// TIA Portal V19 program export: 2 tag tables, 0 data types, 0 data blocks, 5 code blocks (in call order from the OBs), 7 instance data blocks

VAR_GLOBAL   // PLC tag table "Default tag table"
   Sensor_High_High AT %M0.0 : Bool;
   ACK_Alarm_PB AT %M0.1 : Bool;
   Alarm_Reset_PB AT %M0.2 : Bool;
   AlarmStatus AT %M0.3 : Bool;
   Alarm_Acknowledged AT %M0.4 : Bool;
   Alarm_LED AT %M0.5 : Bool;
   Sensor2_High_High AT %M1.0 : Bool;
   AlarmStatus2 AT %M1.1 : Bool;
   Alarm_Acknowledged2 AT %M0.6 : Bool;
   Alarm_LED2 AT %M0.7 : Bool;
END_VAR

VAR_GLOBAL   // PLC tag table "Dispenser_Tags"
   Power_ON AT %M1.0 : Bool;   // Power on Command
   Power_OFF AT %M1.1 : Bool;   // Power off Command
   Power_Active AT %M1.2 : Bool;   // Power is Active
   Start AT %M1.3 : Bool;   // Start Command
   Motor AT %M1.5 : Bool;   // Motor Status
   Gate1 AT %M1.6 : Bool;   // Light Gate Sensor 1
   Gate2 AT %M1.7 : Bool;   // Light Gate Sensor 2
   Gate3 AT %M2.0 : Bool;   // Light Gate Sensor 3
   Gate4 AT %M2.1 : Bool;   // Light Gate Sensor 4
   Gate5 AT %M2.2 : Bool;   // Light Gate Sensor 5
   Dropper_A AT %M2.3 : Bool;   // Dispenser Dropper 1
   Dropper_B AT %M2.4 : Bool;   // Dispenser Dropper 2
   Dropper_C AT %M2.5 : Bool;   // Dispenser Dropper 3
   Stop AT %M1.4 : Bool;   // Stop Command
   SW_A AT %M2.6 : Bool;   // Switch A
   SW_B AT %M2.7 : Bool;   // Switch B
   SW_C AT %M3.0 : Bool;   // Switch C
   Process_Started AT %M3.1 : Bool;   // Dispenser Process Running
   StopDispenser AT %M3.2 : Bool;   // E-Stop for Dispenser
END_VAR

ORGANIZATION_BLOCK "Main"   // OB1, LAD, ProgramCycle
TITLE = "Main Program Sweep (Cycle)"
{ S7_Optimized_Access := 'TRUE' }
// stored: SetENOAutomatically false
   VAR_INPUT
      Initial_Call : Bool;   // Initial call of this OB
      Remanence : Bool;   // =True, if remanent data are available
   END_VAR
BEGIN

REGION Network 1: Sensor 1 - Alarm
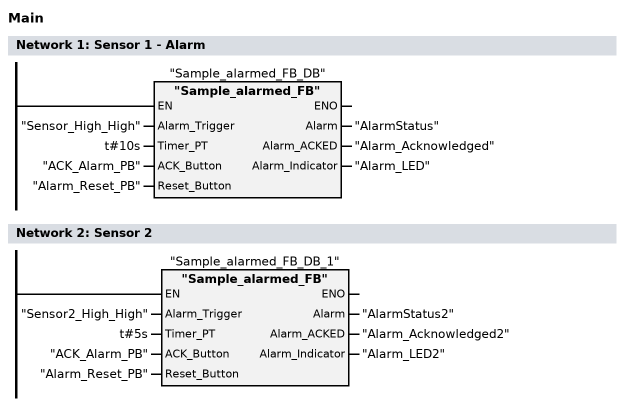
   RUNG wire#powerrail
      "Sample_alarmed_FB_DB"(Alarm_Trigger := "Sensor_High_High", Timer_PT := t#10s, ACK_Button := "ACK_Alarm_PB", Reset_Button := "Alarm_Reset_PB", Alarm => "AlarmStatus", Alarm_ACKED => "Alarm_Acknowledged", Alarm_Indicator => "Alarm_LED")
   END_RUNG
   // the same network as SCL:
   "Sample_alarmed_FB_DB"(Alarm_Trigger := "Sensor_High_High",   // "Sample_alarmed_FB"
                          Timer_PT := t#10s,
                          ACK_Button := "ACK_Alarm_PB",
                          Reset_Button := "Alarm_Reset_PB",
                          Alarm => "AlarmStatus",
                          Alarm_ACKED => "Alarm_Acknowledged",
                          Alarm_Indicator => "Alarm_LED");
END_REGION

REGION Network 2: Sensor 2
   RUNG wire#powerrail
      "Sample_alarmed_FB_DB_1"(Alarm_Trigger := "Sensor2_High_High", Timer_PT := t#5s, ACK_Button := "ACK_Alarm_PB", Reset_Button := "Alarm_Reset_PB", Alarm => "AlarmStatus2", Alarm_ACKED => "Alarm_Acknowledged2", Alarm_Indicator => "Alarm_LED2")
   END_RUNG
   // the same network as SCL:
   "Sample_alarmed_FB_DB_1"(Alarm_Trigger := "Sensor2_High_High",   // "Sample_alarmed_FB"
                           Timer_PT := t#5s,
                           ACK_Button := "ACK_Alarm_PB",
                           Reset_Button := "Alarm_Reset_PB",
                           Alarm => "AlarmStatus2",
                           Alarm_ACKED => "Alarm_Acknowledged2",
                           Alarm_Indicator => "Alarm_LED2");
END_REGION
END_ORGANIZATION_BLOCK

FUNCTION_BLOCK "Sample_alarmed_FB"   // FB1, LAD
TITLE = Alarms -Timed Alarm System
{ S7_Optimized_Access := 'TRUE' }
// stored: MemoryReserve 100, SetENOAutomatically false
   VAR_INPUT
      Alarm_Trigger : Bool;   // Used to Trigger the Alarm Watching
      Timer_PT : Time;   // Time Until Alarm goes off after Trigger
      ACK_Button : Bool;   // Acknowledged Alarm Button
      Reset_Button : Bool;   // Reset Alarm Button
   END_VAR
   VAR_OUTPUT
      Alarm : Bool;   // Current Status of Alarm
      Alarm_ACKED : Bool;   // Alarm Acknowledged (Y/N)
      Alarm_Indicator : Bool;   // Alarm LED Indicator
   END_VAR
   VAR
      Alarm_Timer { S7_SetPoint := 'True'} : TON_TIME;   // Used when Triggering Alarm Active
      Alarm_Timer_Done : Bool;   // Triggers when Alarm Timer Elapsed
      Alarm_Active : Bool;   // Alarm is Active
      Alarm_ACK : Bool;   // Alarm is Acknowledged
      Alarm_Reset : Bool;   // Alarm is Reset
   END_VAR
BEGIN

REGION Network 1: Start Alarm
   // When Alarm_Trigger > Timer_PT the Alarm_Timer is Done
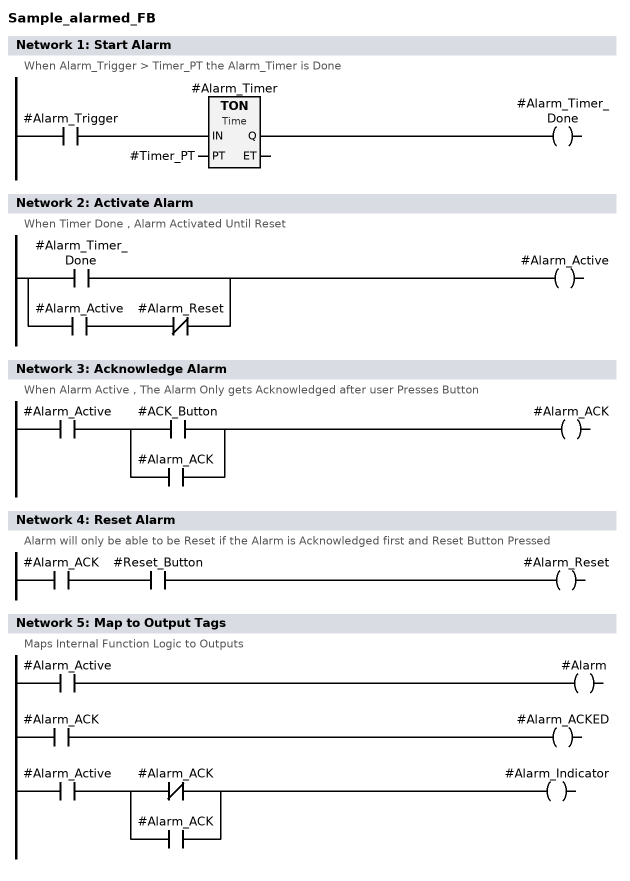
   RUNG wire#powerrail
      Contact( #Alarm_Trigger )
      { S7_Templates := "time_type := Time" } #Alarm_Timer.TON(pt := #Timer_PT, et =>)
      Coil( #Alarm_Timer_Done )
   END_RUNG
   // the same network as SCL:
   #Alarm_Timer(IN := #Alarm_Trigger, PT := #Timer_PT);   // TON
   #Alarm_Timer_Done := #Alarm_Timer.Q;
END_REGION

REGION Network 2: Activate Alarm
   // When Timer Done , Alarm Activated Until Reset
   RUNG wire#powerrail
      Contact( #Alarm_Timer_Done )
      wire#w1
      Coil( #Alarm_Active )
   END_RUNG
   RUNG wire#powerrail
      Contact( #Alarm_Active )
      I_Contact( #Alarm_Reset )
   END_RUNG wire#w1
   // the same network as SCL:
   #Alarm_Active := #Alarm_Timer_Done OR (#Alarm_Active AND NOT #Alarm_Reset);
END_REGION

REGION Network 3: Acknowledge Alarm
   // When Alarm Active , The Alarm Only gets Acknowledged after user Presses Button
   RUNG wire#powerrail
      Contact( #Alarm_Active )
      wire#w1
      Contact( #ACK_Button )
      wire#w2
      Coil( #Alarm_ACK )
   END_RUNG
   RUNG wire#w1
      Contact( #Alarm_ACK )
   END_RUNG wire#w2
   // the same network as SCL:
   #Alarm_ACK := #Alarm_Active AND (#ACK_Button OR #Alarm_ACK);
END_REGION

REGION Network 4: Reset Alarm
   // Alarm will only be able to be Reset if the Alarm is Acknowledged first and Reset Button Pressed
   RUNG wire#powerrail
      Contact( #Alarm_ACK )
      Contact( #Reset_Button )
      Coil( #Alarm_Reset )
   END_RUNG
   // the same network as SCL:
   #Alarm_Reset := #Alarm_ACK AND #Reset_Button;
END_REGION

REGION Network 5: Map to Output Tags
   // Maps Internal Function Logic to Outputs
   RUNG wire#powerrail
      Contact( #Alarm_Active )
      Coil( #Alarm )
   END_RUNG
   RUNG wire#powerrail
      Contact( #Alarm_ACK )
      Coil( #Alarm_ACKED )
   END_RUNG
   RUNG wire#powerrail
      Contact( #Alarm_Active )
      wire#w1
      I_Contact( #Alarm_ACK )
      wire#w2
      Coil( #Alarm_Indicator )
   END_RUNG
   RUNG wire#w1
      Contact( #Alarm_ACK )
   END_RUNG wire#w2
   // the same network as SCL:
   #Alarm := #Alarm_Active;
   #Alarm_ACKED := #Alarm_ACK;
   #Alarm_Indicator := #Alarm_Active AND (NOT #Alarm_ACK OR #Alarm_ACK);
END_REGION

REGION Network 6: Spare
END_REGION
END_FUNCTION_BLOCK

FUNCTION_BLOCK "Alarm_Trigger"   // FB2, LAD
TITLE = Emergency Stop / Alarm
{ S7_Optimized_Access := 'TRUE' }
// Will Hold Info On Alarms and Reset
// stored: MemoryReserve 100, SetENOAutomatically false
   VAR_INPUT
      Alarm_Trigger : Bool;   // Input that Triggers Alarm
      Timer_PT : Time;   // Timer for Trigger Set
      Ack_PB : Bool;   // Acknowledge Alarm Button
      Reset_PB : Bool;   // Reset Alarm Button
   END_VAR
   VAR_OUTPUT
      ALARM : Bool;   // Alarm Status
      ALARM_ACKED : Bool;   // Alarm Acknowledge Status
      ALARM_BLINK : Bool;   // Alarm LED Status
   END_VAR
   VAR
      Alarm_TD : Bool;   // Alarm was Triggered
      Alarm_Active : Bool;   // Alarm is Active
      Alarm_ACK : Bool;   // Alarm was Acknowledged
      Alarm_Reset : Bool;   // Alarm was Reset
      Alarm_Timer { S7_SetPoint := 'True'} : TON_TIME;   // Alarm Timer
   END_VAR
BEGIN

REGION Network 1: Alarm Triggers ( After holding for PTime)
   // Sets Alarm to Triggered after some time.
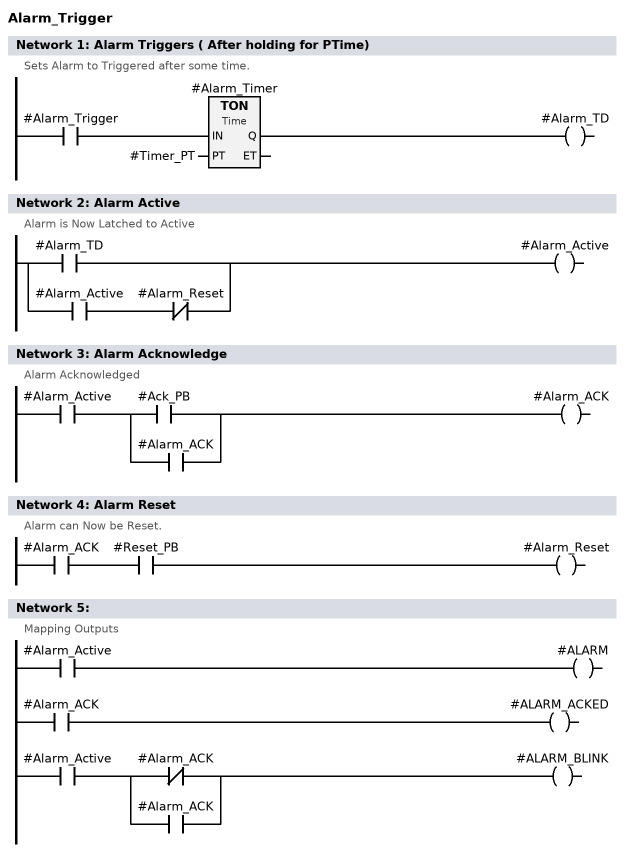
   RUNG wire#powerrail
      Contact( #Alarm_Trigger )
      { S7_Templates := "time_type := Time" } #Alarm_Timer.TON(pt := #Timer_PT, et =>)
      Coil( #Alarm_TD )
   END_RUNG
   // the same network as SCL:
   #Alarm_Timer(IN := #Alarm_Trigger, PT := #Timer_PT);   // TON
   #Alarm_TD := #Alarm_Timer.Q;
END_REGION

REGION Network 2: Alarm Active
   // Alarm is Now Latched to Active
   RUNG wire#powerrail
      Contact( #Alarm_TD )
      wire#w1
      Coil( #Alarm_Active )
   END_RUNG
   RUNG wire#powerrail
      Contact( #Alarm_Active )
      I_Contact( #Alarm_Reset )
   END_RUNG wire#w1
   // the same network as SCL:
   #Alarm_Active := #Alarm_TD OR (#Alarm_Active AND NOT #Alarm_Reset);
END_REGION

REGION Network 3: Alarm Acknowledge
   // Alarm Acknowledged
   RUNG wire#powerrail
      Contact( #Alarm_Active )
      wire#w1
      Contact( #Ack_PB )
      wire#w2
      Coil( #Alarm_ACK )
   END_RUNG
   RUNG wire#w1
      Contact( #Alarm_ACK )
   END_RUNG wire#w2
   // the same network as SCL:
   #Alarm_ACK := #Alarm_Active AND (#Ack_PB OR #Alarm_ACK);
END_REGION

REGION Network 4: Alarm Reset
   // Alarm can Now be Reset.
   RUNG wire#powerrail
      Contact( #Alarm_ACK )
      Contact( #Reset_PB )
      Coil( #Alarm_Reset )
   END_RUNG
   // the same network as SCL:
   #Alarm_Reset := #Alarm_ACK AND #Reset_PB;
END_REGION

REGION Network 5
   // Mapping Outputs
   RUNG wire#powerrail
      Contact( #Alarm_Active )
      Coil( #ALARM )
   END_RUNG
   RUNG wire#powerrail
      Contact( #Alarm_ACK )
      Coil( #ALARM_ACKED )
   END_RUNG
   RUNG wire#powerrail
      Contact( #Alarm_Active )
      wire#w1
      I_Contact( #Alarm_ACK )
      wire#w2
      Coil( #ALARM_BLINK )
   END_RUNG
   RUNG wire#w1
      Contact( #Alarm_ACK )
   END_RUNG wire#w2
   // the same network as SCL:
   #ALARM := #Alarm_Active;
   #ALARM_ACKED := #Alarm_ACK;
   #ALARM_BLINK := #Alarm_Active AND (NOT #Alarm_ACK OR #Alarm_ACK);
END_REGION

REGION Network 6: Spare Network
END_REGION
END_FUNCTION_BLOCK

FUNCTION_BLOCK "Analogue_Input_HMI"   // FB5, LAD
TITLE = Adjust Level Meter From HMI to Control Pump Simulation
{ S7_Optimized_Access := 'TRUE' }
// stored: MemoryReserve 100, SetENOAutomatically false
   VAR_INPUT
      Sensor_Reading { ExternalAccessible := 'False'; ExternalVisible := 'False'; ExternalWritable := 'False'} : Int;   // Reading from Sensor ( on HMI)
   END_VAR
   VAR_OUTPUT
      High_LVL { ExternalAccessible := 'False'; ExternalVisible := 'False'; ExternalWritable := 'False'} : Bool;   // Level High Reached
      Sensor_Reading_Real { ExternalAccessible := 'False'; ExternalVisible := 'False'; ExternalWritable := 'False'} : Real;   // Reading from Sensor (Real)
      Low_LVL { ExternalAccessible := 'False'; ExternalVisible := 'False'; ExternalWritable := 'False'} : Bool;   // Level Low Reached
   END_VAR
   VAR_IN_OUT
      Level_High_SP { ExternalAccessible := 'False'; ExternalVisible := 'False'; ExternalWritable := 'False'} : Real;   // High Level Setpoint Value
      Level_Low_SP { ExternalAccessible := 'False'; ExternalVisible := 'False'; ExternalWritable := 'False'} : Real;   // Low Level Setpoint Value
   END_VAR
BEGIN

REGION Network 1: Convert Int to Real
   // Basic Conversion
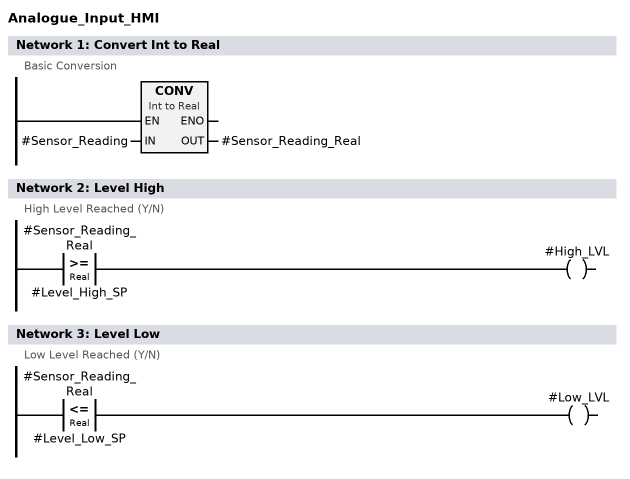
   RUNG wire#powerrail
      { S7_Templates := "[SrcType := Int, DestType := Real]" } Convert(in := #Sensor_Reading, out => #Sensor_Reading_Real)
   END_RUNG
   // the same network as SCL:
   #Sensor_Reading_Real := INT_TO_REAL(#Sensor_Reading);
END_REGION

REGION Network 2: Level High
   // High Level Reached (Y/N)
   RUNG wire#powerrail
      { S7_Templates := "SrcType := Real" } GE_Contact(in1 := #Sensor_Reading_Real, in2 := #Level_High_SP)
      Coil( #High_LVL )
   END_RUNG
   // the same network as SCL:
   #High_LVL := #Sensor_Reading_Real >= #Level_High_SP;
END_REGION

REGION Network 3: Level Low
   // Low Level Reached (Y/N)
   RUNG wire#powerrail
      { S7_Templates := "SrcType := Real" } LE_Contact(in1 := #Sensor_Reading_Real, in2 := #Level_Low_SP)
      Coil( #Low_LVL )
   END_RUNG
   // the same network as SCL:
   #Low_LVL := #Sensor_Reading_Real <= #Level_Low_SP;
END_REGION

REGION Network 4: Spare Network
END_REGION
END_FUNCTION_BLOCK

FUNCTION_BLOCK "Pump_Block"   // FB4, LAD
TITLE = Pump Block
{ S7_Optimized_Access := 'TRUE' }
// Function Block for Pumps
// stored: MemoryReserve 100, SetENOAutomatically false
   VAR_INPUT
      Mode_Selection : Bool;   // Auto or Manual Mode Selected
      Start_Manual : Bool;   // Starting by Manual
      Stop_Manual : Bool;   // Stopping by Manual
      Start_Auto : Bool;   // Starting by Auto
      Stop_Auto : Bool;   // Stopping by Auto
      Level_High : Bool;   // Level High Alarm
      Level_Low : Bool;   // Level Low Alarm
      Set_Time_Start : DInt;   // Setting Timer for Start Auto
      Overload : Bool;   // Motor Overload
      Reset_Fault : Bool;   // Reset Fault Command
   END_VAR
   VAR_OUTPUT
      Pump_Run : Bool;   // Motor Started
      Fault : Bool;   // Motor Fault
      Running_Auto_Mode : Bool;   // Running Auto Mode Signal
   END_VAR
   VAR
      Timer_Start : IEC_TIMER;   // Starting Timer for Auto Mode
      Start_Auto_Activated : Bool;   // Starting Auto Activated
   END_VAR
   VAR_TEMP
      Timer_Start_Output : Bool;   // Output of Timer Started
   END_VAR
   VAR_TEMP   // added for the SCL form of the ladder/FBD networks
      _w1 : Bool;
   END_VAR
BEGIN

REGION Network 1: Motor overload Interlocking
   // If Overloaded trigger a fault
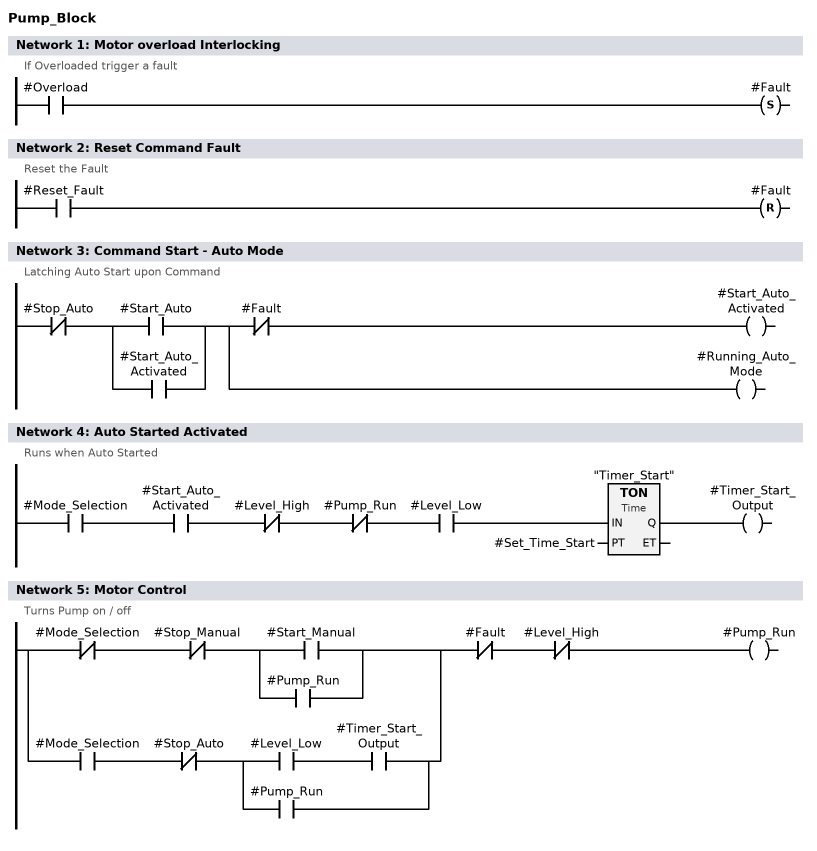
   RUNG wire#powerrail
      Contact( #Overload )
      S_Coil( #Fault )
   END_RUNG
   // the same network as SCL:
   IF #Overload THEN #Fault := TRUE; END_IF;
END_REGION

REGION Network 2: Reset Command Fault
   // Reset the Fault
   RUNG wire#powerrail
      Contact( #Reset_Fault )
      R_Coil( #Fault )
   END_RUNG
   // the same network as SCL:
   IF #Reset_Fault THEN #Fault := FALSE; END_IF;
END_REGION

REGION Network 3: Command Start - Auto Mode
   // Latching Auto Start upon Command
   RUNG wire#powerrail
      I_Contact( #Stop_Auto )
      wire#w1
      Contact( #Start_Auto )
      wire#w2
      I_Contact( #Fault )
      Coil( #Start_Auto_Activated )
   END_RUNG
   RUNG wire#w1
      Contact( #Start_Auto_Activated )
   END_RUNG wire#w2
   RUNG wire#w2
      Coil( #Running_Auto_Mode )
   END_RUNG
   // the same network as SCL:
   #_w1 := NOT #Stop_Auto AND (#Start_Auto OR #Start_Auto_Activated);
   #Start_Auto_Activated := #_w1 AND NOT #Fault;
   #Running_Auto_Mode := #_w1;
END_REGION

REGION Network 4: Auto Started Activated
   // Runs when Auto Started
   RUNG wire#powerrail
      Contact( #Mode_Selection )
      Contact( #Start_Auto_Activated )
      I_Contact( #Level_High )
      I_Contact( #Pump_Run )
      Contact( #Level_Low )
      { S7_Templates := "time_type := Time" } "Timer_Start".TON(pt := #Set_Time_Start, et =>)
      Coil( #Timer_Start_Output )
   END_RUNG
   // the same network as SCL:
   "Timer_Start".TON(IN := #Mode_Selection AND #Start_Auto_Activated AND NOT #Level_High AND NOT #Pump_Run AND #Level_Low,
                     PT := #Set_Time_Start);
   #Timer_Start_Output := "Timer_Start".Q;
END_REGION

REGION Network 5: Motor Control
   // Turns Pump on / off
   RUNG wire#powerrail
      I_Contact( #Mode_Selection )
      I_Contact( #Stop_Manual )
      wire#w1
      Contact( #Start_Manual )
      wire#w2
      I_Contact( #Fault )
      I_Contact( #Level_High )
      Coil( #Pump_Run )
   END_RUNG
   RUNG wire#w1
      Contact( #Pump_Run )
   END_RUNG wire#w2
   RUNG wire#powerrail
      Contact( #Mode_Selection )
      I_Contact( #Stop_Auto )
      wire#w3
      Contact( #Level_Low )
      Contact( #Timer_Start_Output )
   END_RUNG wire#w2
   RUNG wire#w3
      Contact( #Pump_Run )
   END_RUNG wire#w2
   // the same network as SCL:
   #Pump_Run := ((NOT #Mode_Selection AND NOT #Stop_Manual AND (#Start_Manual OR #Pump_Run)) OR (#Mode_Selection AND NOT #Stop_Auto AND ((#Level_Low AND #Timer_Start_Output) OR #Pump_Run))) AND NOT #Fault AND NOT #Level_High;
END_REGION

REGION Network 6: Spare Network
END_REGION
END_FUNCTION_BLOCK

DATA_BLOCK "Sample_alarmed_FB_DB"   // DB1
// stored: InstanceOfName Sample_alarmed_FB, InstanceOfType FB
"Sample_alarmed_FB"
BEGIN
END_DATA_BLOCK

DATA_BLOCK "Sample_alarmed_FB_DB_1"   // DB2
// stored: InstanceOfName Sample_alarmed_FB, InstanceOfType FB
"Sample_alarmed_FB"
BEGIN
END_DATA_BLOCK

DATA_BLOCK "Alarm_No1"   // DB6
// stored: InstanceOfName Alarm_Trigger, InstanceOfType FB
"Alarm_Trigger"
BEGIN
END_DATA_BLOCK

DATA_BLOCK "Mixer_Block_DB"   // DB5
// stored: InstanceOfName Mixer_Block, InstanceOfType FB
"Mixer_Block"
BEGIN
END_DATA_BLOCK

DATA_BLOCK "T_Dropper_A"   // DB1
{ S7_Optimized_Access := 'TRUE' }
// stored: InstanceOfName IEC_TIMER, OfSystemLibElement IEC_TIMER, OfSystemLibVersion 1.0
"IEC_TIMER"
   // VAR
   //    PT : Time;
   //    ET { ExternalWritable := 'False'} : Time;
   //    IN : Bool;
   //    Q { ExternalWritable := 'False'} : Bool;
   // END_VAR
BEGIN
END_DATA_BLOCK

DATA_BLOCK "T_Dropper_B"   // DB2
{ S7_Optimized_Access := 'TRUE' }
// stored: InstanceOfName IEC_TIMER, OfSystemLibElement IEC_TIMER, OfSystemLibVersion 1.0
"IEC_TIMER"
   // VAR
   //    PT : Time;
   //    ET { ExternalWritable := 'False'} : Time;
   //    IN : Bool;
   //    Q { ExternalWritable := 'False'} : Bool;
   // END_VAR
BEGIN
END_DATA_BLOCK

DATA_BLOCK "T_Dropper_C"   // DB3
{ S7_Optimized_Access := 'TRUE' }
// stored: InstanceOfName IEC_TIMER, OfSystemLibElement IEC_TIMER, OfSystemLibVersion 1.0
"IEC_TIMER"
   // VAR
   //    PT : Time;
   //    ET { ExternalWritable := 'False'} : Time;
   //    IN : Bool;
   //    Q { ExternalWritable := 'False'} : Bool;
   // END_VAR
BEGIN
END_DATA_BLOCK
